(* Schneider Machine Expert - Basic project test1, file version 2.0.0.0 *)
(* ProjectInformations: Name=New project *)

HARDWARE
  Cpu 0: TM221CE16R
  EthernetConfiguration: NetworkName=M221, IpAllocationMode=FixedAddress, IpAddress=0.0.0.0, SubnetMask=0.0.0.0
  SerialLineConfiguration: Baud=Baud19200, Parity=ParityEven, DataBits=DataBits8, StopBits=StopBits1, PhysicalMedium=PhysicalMediumRs485, TransmissionMode=TransmissionModeModbusRtu, SlaveId=1, Addressing=SlaveAddressing
  MastTask: UsePeriodScanMode=false, PeriodScan=100
  FastTask: Period=255
  CpuBehavior: StartingMode=StartAsPreviousState, AutoSaveRamOnEeprom=true, WatchdogPeriod=250

SYMBOLS  (address, symbol, comment, settings)

POU New POU
  (* SectionNumber=1 *)

// Rung 0
  LD %I0.1
  AND %I0.8
  ST %M1
  // as ST:
  //   %M1 := %I0.1 AND %I0.8;

// Rung 1
  LD %M5
  AND %M259
  ST %M260
  // as ST:
  //   %M260 := %M5 AND %M259;

// Rung 2
  LD %M307
  ST %M498
  // as ST:
  //   %M498 := %M307;
